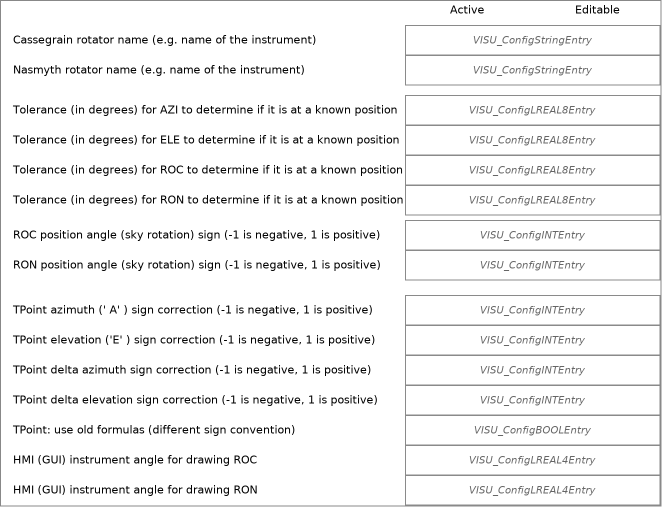
VISUALIZATION VISU_AxesConfig_General  // 662x507
VAR_IN_OUT
    editable : AxesConfig;
	active : AxesConfig;
END_VAR
    Frame (405,25 255x30)
        shows VISU_ConfigStringEntry(active := active.cassegrainRotatorName, editable := editable.cassegrainRotatorName)
    Label (405,0 125x20), "Active"
    Label (535,0 125x20), "Editable"
    Label (10,25 370x30), "Cassegrain rotator name (e.g. name of the instrument)"
    Frame (405,55 255x30)
        shows VISU_ConfigStringEntry(active := active.nasmythRotatorName, editable := editable.nasmythRotatorName)
    Label (10,55 370x30), "Nasmyth rotator name (e.g. name of the instrument)"
    Frame (405,95 255x30)
        shows VISU_ConfigLREAL8Entry(active := active.knownPositionToleranceAzi, editable := editable.knownPositionToleranceAzi)
    Label (10,95 395x30), "Tolerance (in degrees) for AZI to determine if it is at a known position"
    Label (10,125 395x30), "Tolerance (in degrees) for ELE to determine if it is at a known position"
    Frame (405,125 255x30)
        shows VISU_ConfigLREAL8Entry(active := active.knownPositionToleranceEle, editable := editable.knownPositionToleranceEle)
    Label (10,155 395x30), "Tolerance (in degrees) for ROC to determine if it is at a known position"
    Frame (405,155 255x30)
        shows VISU_ConfigLREAL8Entry(active := active.knownPositionToleranceRoc, editable := editable.knownPositionToleranceRoc)
    Label (10,185 395x30), "Tolerance (in degrees) for RON to determine if it is at a known position"
    Frame (405,185 255x30)
        shows VISU_ConfigLREAL8Entry(active := active.knownPositionToleranceRon, editable := editable.knownPositionToleranceRon)
    Frame (405,295 255x30)
        shows VISU_ConfigINTEntry(active := active.tpointAziSign, editable := editable.tpointAziSign)
    Label (10,295 395x30), "TPoint azimuth (' A' ) sign correction (-1 is negative, 1 is positive)"
    Frame (405,325 255x30)
        shows VISU_ConfigINTEntry(active := active.tpointEleSign, editable := editable.tpointEleSign)
    Label (10,325 395x30), "TPoint elevation ('E' ) sign correction (-1 is negative, 1 is positive)"
    Frame (405,355 255x30)
        shows VISU_ConfigINTEntry(active := active.tpointDeltaAziSign, editable := editable.tpointDeltaAziSign)
    Label (10,355 395x30), "TPoint delta azimuth sign correction (-1 is negative, 1 is positive)"
    Frame (405,385 255x30)
        shows VISU_ConfigINTEntry(active := active.tpointDeltaEleSign, editable := editable.tpointDeltaEleSign)
    Label (10,385 395x30), "TPoint delta elevation sign correction (-1 is negative, 1 is positive)"
    Label (10,415 395x30), "TPoint: use old formulas (different sign convention)"
    Frame (405,415 255x30)
        shows VISU_ConfigBOOLEntry(active := active.tpointOldFormulas, editable := editable.tpointOldFormulas)
    Frame (405,220 255x30)
        shows VISU_ConfigINTEntry(active := active.rocPositionAngleSign, editable := editable.rocPositionAngleSign)
    Label (10,220 395x30), "ROC position angle (sky rotation) sign (-1 is negative, 1 is positive)"
    Frame (405,250 255x30)
        shows VISU_ConfigINTEntry(active := active.ronPositionAngleSign, editable := editable.ronPositionAngleSign)
    Label (10,250 395x30), "RON position angle (sky rotation) sign (-1 is negative, 1 is positive)"
    Frame (405,445 255x30)
        shows VISU_ConfigLREAL4Entry(active := active.rocGuiAngle, editable := editable.rocGuiAngle)
    Label (10,445 395x30), "HMI (GUI) instrument angle for drawing ROC"
    Frame (405,475 255x30)
        shows VISU_ConfigLREAL4Entry(active := active.ronGuiAngle, editable := editable.ronGuiAngle)
    Label (10,475 395x30), "HMI (GUI) instrument angle for drawing RON"
END_VISUALIZATION

(* stored: Version 1.1.0.1, ProductVersion 3.1.4019.2
   Visu VISU_AxesConfig_General: Id {aa99e4fa-c602-4fd0-af6f-d43562985fa0} *)
